(* CoDeSys 2.3.9.47 project: bms.pro *)
(* Libraries: WagoCANopen_02.lib 16.5.13 13:00:50, WagoCANLayer2_02.lib 23.6.14 12:08:28, Standard.lib 20.5.14 07:13:26, Iecsfc.lib 16.5.13 13:00:50, SYSLIBCALLBACK.LIB 16.5.13 13:00:50 *)

(* PLC configuration (modules and I/O channels)
0750-0430 8 DI 24 V DC 3.0ms [Type_1_8_Channels] node 0, in %IB0 out %QB0
  AT %IX0.0 [BOOLOnX_I] Ch_1 Digital input
  AT %IX0.1 [BOOLOnX_I] Ch_2 Digital input
  AT %IX0.2 [BOOLOnX_I] Ch_3 Digital input
  AT %IX0.3 [BOOLOnX_I] Ch_4 Digital input
  AT %IX0.4 [BOOLOnX_I] Ch_5 Digital input
  AT %IX0.5 [BOOLOnX_I] Ch_6 Digital input
  AT %IX0.6 [BOOLOnX_I] Ch_7 Digital input
  AT %IX0.7 [BOOLOnX_I] Ch_8 Digital input
Modbus variables [PFC200MODBUS] node 1, in %IB0 out %QB0 {PlcStopBehaviour = 1; FiledbusErrorBehaviour = 1; TcpOperation = 1; TcpPort = 502; TcpTimeout = 600; UdpOperation = 1; UdpPort = 502; RtuOperation = 0; NodeId = 1; ResponseTimeout = 5000; Interface = 0; Baud = 115200; StopBits = 1; Parity = 1; FlowCtrl = 0; PhysInterface = 0}
CANopen-Master [CanMaster] node 2, in %IB6000 out %QB6000
Modbus-Master [MB_MASTER] node 3, in %IB0 out %QB0
*)

(* Task configuration *)
TASK t500 (PRIORITY := 29, INTERVAL := T#500ms);
	PLC_PRG();
END_TASK
TASK Open (PRIORITY := 31, SINGLE := canStart);
	OPEN_CAN();
END_TASK
TASK Close (PRIORITY := 30, SINGLE := canStop);
	CLOSE_CAN();
END_TASK

(* Global variable list: Globale_Variablen *)
VAR_GLOBAL
	FRAME:BOOL;
	canStart:BOOL := FALSE;
	canStop:BOOL := FALSE;
	canOpen : CAN_OPEN;
	canClose:CAN_CLOSE;
END_VAR

(* POU PLC_PRG, ST *)
PROGRAM PLC_PRG
VAR
	canReset:CAN_RESET;
	canLedSet:CAN_SET_LED;

	canId:WORD;
	can11BitFrame :CAN_RX_11BIT_FRAME;
	TON1:TON;
END_VAR
(*canReset(ENABLE := TRUE);*)
(*canOpen(BAUDRATE := 500000 ,ENABLE := TRUE );*)

(*TON1(IN := NOT  frame ,  PT := T#0.1s);
frame := TON1.Q;*)

(*canLedSet(MODE:= LED_OP , ENABLE:= TRUE);*)

canId := 16#381;

can11BitFrame(
		CAN_ID:= canId,
		CAN_BUFFER:= FALSE,
		ENABLE := TRUE,
		READ_FRAME:= FRAME
	);

(*IF canOpen.CONFIRM = TRUE THEN
	can11BitFrame(
		CAN_ID:= canId,
		CAN_BUFFER:= FALSE,
		ENABLE := TRUE,
		READ_FRAME:= FRAME
	);
END_IF*)

(*frame := NOT frame;*)
END_PROGRAM

(* POU OPEN_CAN, ST *)
PROGRAM OPEN_CAN
VAR
END_VAR
canOpen.BAUDRATE :=500000;
canOpen.ENABLE := TRUE;
canStop := FALSE;
canClose.ENABLE := FALSE;
END_PROGRAM

(* POU CLOSE_CAN, ST *)
PROGRAM CLOSE_CAN
VAR
END_VAR
canClose.ENABLE := TRUE;
canStart := FALSE;
canOpen.ENABLE := FALSE;
END_PROGRAM

(* POU toggle, ST *)
PROGRAM toggle
VAR
END_VAR
;
END_PROGRAM

(* Visualisation CAN_VISU
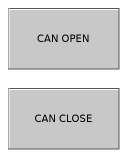
button at (70,40)-(181,101): text "CAN OPEN"; runs INTERN ASSIGN canStart:=(TRUE)
button at (70,120)-(181,181): text "CAN CLOSE"; runs INTERN ASSIGN canStop:=(TRUE)
*)
